# EPICS substitutions: EUROTHRM/EUROTHRM-IOC-01App/Db/devEurothrmA05.substitutions
# Note: this file is generated by generate_substitutions.py
file devEurothrm.template {
pattern { P, GAD, LAD, MODBUS_PV, MODBUS_SP, MODBUS_P, MODBUS_I, MODBUS_D, MODBUS_HS, MODBUS_LS, MODBUS_AT, MODBUS_HO, MODBUS_OP }
{ "\$(P)", "0", "5", "4097", "4098", "4102", "4104", "4105", "4207", "4208", "4366", "4126", "4099" }
}
